Staubli VAL3: listadd.pgx

public program listAdd(string& x_sItems[])
  local num i
  local num l_nSize
begin
  //Header begin
  //Description of program
  //  Insert x_sItems into the list.
  //
  //Input parameters
  //  string x_sItems :
  //    role : Items to add
  //
  //Example
  //  call listAdd("Name: > ")
  //
  //History
  //  Creation : 28-04-08 - f.Rob
  //Header end
  for i=0 to (size(x_sItems)-1)
    if (size(sItems)!=1 or sItems!="") and x_sItems[i]!=""
      //Insert an Item in sItems[] after the last element.
      insert(sItems[size(sItems)])
      //Insert an Item in bReadWrite[] after the last element.
      insert(bReadWrite[size(bReadWrite)])
    endIf
    if x_sItems[i]!=""
      sItems[size(sItems)-1]=x_sItems[i]
      //For default the RW is true
      bReadWrite[size(bReadWrite)-1]=true
    endIf
  endFor
end
